TYPE
    EtcMasterBase_62654B43 :
    STRUCT
    END_STRUCT
END_TYPE

(* stored: Version 1.1.0.1, ProductVersion 3.1.4024.12
   DUT EtcMasterBase_62654B43: Id {d13a95a4-d79f-0603-37d5-c6831f240e9d} *)
